FUNCTION_BLOCK FB_AxisStatus_TestDouble IMPLEMENTS I_AxisStatus
VAR_INPUT
END_VAR
VAR_OUTPUT
END_VAR
VAR
END_VAR

{warning 'Add property implementation'}
PROPERTY Aborted : BOOL
GET
END_GET
END_PROPERTY

{warning 'Add property implementation'}
PROPERTY Active : BOOL
GET
END_GET
END_PROPERTY

{warning 'Add method implementation '}
METHOD AxisEnabled : BOOL
END_METHOD

{warning 'Add property implementation'}
PROPERTY AxisID : UDINT
GET
END_GET
END_PROPERTY

{warning 'Add property implementation'}
PROPERTY AxisState : MC_AxisStates
GET
END_GET
END_PROPERTY

{warning 'Add property implementation'}
PROPERTY Busy : BOOL
GET
END_GET
END_PROPERTY

{warning 'Add property implementation'}
PROPERTY Done : BOOL
GET
END_GET
END_PROPERTY

{warning 'Add property implementation'}
PROPERTY Error : BOOL
GET
END_GET
END_PROPERTY

{warning 'Add property implementation'}
PROPERTY ErrorID : UDINT
GET
END_GET
END_PROPERTY

{warning 'Add property implementation'}
PROPERTY InTargetPosition : BOOL
GET
END_GET
END_PROPERTY

{warning 'Add property implementation'}
PROPERTY MeasuredAcceleration : LREAL
GET
END_GET
END_PROPERTY

{warning 'Add property implementation'}
PROPERTY MeasuredPosition : LREAL
GET
END_GET
END_PROPERTY

{warning 'Add property implementation'}
PROPERTY MeasuredPositionDiff : LREAL
GET
END_GET
END_PROPERTY

{warning 'Add property implementation'}
PROPERTY MeasuredVelocity : LREAL
GET
END_GET
END_PROPERTY

{warning 'Add property implementation'}
PROPERTY Message : T_MAXSTRING
GET
END_GET
END_PROPERTY

{warning 'Add property implementation'}
PROPERTY NegativeMotionIsEnabled : BOOL
GET
END_GET
END_PROPERTY

{warning 'Add property implementation'}
PROPERTY PositiveMotionIsEnabled : BOOL
GET
END_GET
END_PROPERTY

{warning 'Add property implementation'}
PROPERTY StandStill : BOOL
GET
END_GET
END_PROPERTY

{warning 'Add property implementation'}
PROPERTY Stopped : BOOL
GET
END_GET
END_PROPERTY

END_FUNCTION_BLOCK

(* stored: Version 1.1.0.1
   POU FB_AxisStatus_TestDouble: Id {3bc600b5-957e-4849-b712-96877efc6ba9}, SpecialFunc None
   Property Aborted: Id {1cd080ba-bc33-4e34-957d-6be955fba72e}
   Get Get: Id {704de71e-6cbb-4217-a018-a3cc3bb90377}
   Property Active: Id {bcbcd1f5-9bdd-483e-8957-a6b5b966ad19}
   Get Get: Id {f2b4eb49-2334-4872-ac07-9f23aec27a72}
   Method AxisEnabled: Id {9aae6fac-ee07-4c85-882c-620886cbadd4}
   Property AxisID: Id {bff40ee1-06b1-4df0-92bc-bfd115d5e98a}
   Get Get: Id {292cf9ef-eda5-4fcb-b12c-b9c346d79e1d}
   Property AxisState: Id {ebb97ecd-8e11-4182-9b1b-5faf014bb5a1}
   Get Get: Id {b5470e90-2038-4e61-8610-b3c18930ad80}
   Property Busy: Id {a5ce5183-3c89-4068-b8c3-1c528ab5cc11}
   Get Get: Id {4b26e38d-9851-4f5b-bcad-e13a6c4f8a2d}
   Property Done: Id {7e8fb5a9-d15f-4828-be4c-9dd4fdc846e7}
   Get Get: Id {87fb51ee-c745-49e1-b352-a346dc7a760a}
   Property Error: Id {6cba1b11-1226-4cb0-987c-89386c0483d6}
   Get Get: Id {b46f2816-361f-4cf4-be17-9d564e98b7f5}
   Property ErrorID: Id {3d7891e3-0208-4311-b802-65987052746a}
   Get Get: Id {341bf391-9f2d-4b4e-bea0-08f2991226c9}
   Property InTargetPosition: Id {7438218c-d7f7-4cd1-a9d9-a059e55b26a5}
   Get Get: Id {2cc0771c-d5b5-4348-bbe3-eb59256647e7}
   Property MeasuredAcceleration: Id {dda5b53f-b549-44bd-a948-0cf0cca437da}
   Get Get: Id {61b16222-d9bd-46c0-9d39-b633f20338fe}
   Property MeasuredPosition: Id {c4db3336-33eb-4da1-a007-b013e850f1b6}
   Get Get: Id {3cf9170f-548b-4b74-a108-559ddb84c33b}
   Property MeasuredPositionDiff: Id {48904782-d7b3-49d8-8c29-1f61cb7a25eb}
   Get Get: Id {a76a61b2-db76-4286-866a-0579aadbd033}
   Property MeasuredVelocity: Id {9bafa369-3599-46c7-89ff-74cc0455a05d}
   Get Get: Id {1fa48a9c-9bb4-4acc-811e-339f02b75a6c}
   Property Message: Id {dfc18d57-d39c-4797-9061-fb566f1326fb}
   Get Get: Id {b2efc810-d05a-4cae-aefa-93c438f5bef4}
   Property NegativeMotionIsEnabled: Id {351fee6f-98e4-4b2f-af5b-727682450935}
   Get Get: Id {7a83df16-ddb4-4d27-b4c7-b9d6cdb6577c}
   Property PositiveMotionIsEnabled: Id {681ceff0-67cb-4abb-8400-ff6cb310f3b9}
   Get Get: Id {4c689123-8e51-4deb-bee2-46445194aaf0}
   Property StandStill: Id {a8a6b632-0e1f-4eee-8917-08fc6e7ed16c}
   Get Get: Id {0f587b3c-d976-4bd8-abf8-7ce160a5267a}
   Property Stopped: Id {0b2d656e-b71d-4260-ab28-2263e2b7d51a}
   Get Get: Id {f59a4de3-7373-46f6-b9e3-9447f329aa63} *)
